// TIA Portal V20 export
TYPE "typeCmInterface"
// stored: Access Published, Namespace Unit1.Em4
   STRUCT
      softcam : "Unit1.Em4.typeCmInterfaceSoftCam";
      brakeTest : "Unit1.Em4.typeCmInterfaceBrakeTest";
   END_STRUCT;
END_TYPE
